FUNCTION_BLOCK MockLogger IMPLEMENTS I_TraceLogger
VAR
	_CallCount : UINT;
	_LastSource : T_MaxString;
	_LastMessage : T_MaxString;
	_LastSeverity : UINT;
END_VAR

PROPERTY CallCount : UINT
GET
CallCount := _CallCount;
END_GET
END_PROPERTY

PROPERTY LastMessage : T_Maxstring
GET
LastMessage := _LastMessage;
END_GET
END_PROPERTY

PROPERTY LastSeverity : UINT
GET
LastSeverity := _LastSeverity;
END_GET
END_PROPERTY

PROPERTY LastSource : T_Maxstring
GET
LastSource := _LastSource;
END_GET
END_PROPERTY

METHOD LogMessage
VAR_INPUT
	Key	: Base_Library.T_MaxString;
	Value	: Base_Library.T_MaxString;
	SourceId	: UDINT := 0;
	TimeStamp	: ULINT := 0;
	MessageId	: UDINT := 1;
	Severity	: USINT := 1;
END_VAR
_CallCount := _CallCount + 1;

_LastSource := key;

_LastMessage := value;

_LastSeverity := Severity;
END_METHOD

END_FUNCTION_BLOCK

(* stored: Version 1.1.0.1
   POU MockLogger: Id {935a9ae7-99c4-4d7b-827e-2cc299904c5b}, SpecialFunc None
   Property CallCount: Id {0ff265de-654f-4905-803d-b3ce4350e914}
   Get Get: Id {52d92ede-2d3d-4757-a13a-85da389f246d}
   Property LastMessage: Id {c51bb7f5-3cb3-44cd-a88c-9cef155bd592}
   Get Get: Id {0f1ff1b1-b5ea-46c7-94b0-1bb304f8757b}
   Property LastSeverity: Id {8b633f05-ead0-46c7-96da-6dd0ef241d5d}
   Get Get: Id {2f9784d6-c997-4286-8055-0418e465f54c}
   Property LastSource: Id {34343b50-6d80-47b9-8442-2ca273213668}
   Get Get: Id {3d25db67-9c70-4815-8de8-b2be1ec087d4}
   Method LogMessage: Id {4772d697-6dac-4b50-8905-8c66516f5071} *)
